TYPE TcoUrRoboticsT2OBitRegs :
STRUCT
	{attribute addProperty Name "<#Bit registers#>"}
	Register : ARRAY[0..63] OF BOOL;
END_STRUCT
END_TYPE

(* stored: Version 1.1.0.1, ProductVersion 3.1.4024.12
   DUT TcoUrRoboticsT2OBitRegs: Id {f838210b-aaae-0d17-1ed7-533f8c40d546} *)
